# EPICS substitutions: ion_ps/ion_psApp/Db/ion_ps.substitutions
file kri_rf.template { pattern
{ Sys	, Dev		, PORT		}
{ Depo	, "{PS:1}"	, Depo_PS1	}
}
